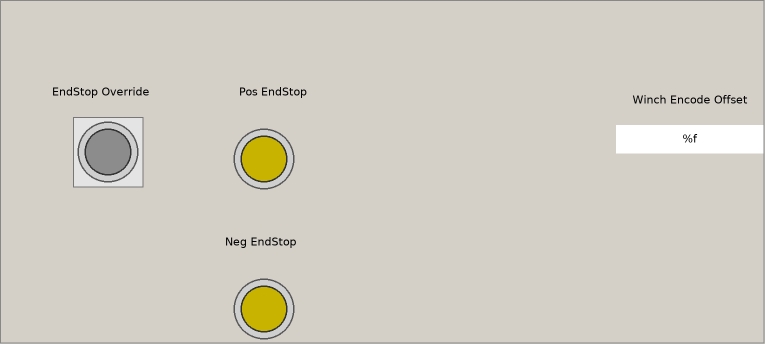
VISUALIZATION HMI  // 765x344
    PushSwitch (73,117 70x70), variable: HMI.bEndStopOverride, behaviour: TOGGLE, style: Switch-PushSwitch-Gray
    Lamp1 (229,124 70x70), variable: P_Outputs.bEndStopPosActive, style: Lamp-Lamp1-Yellow
    Label (26,77 150x30), "EndStop Override"
    Label (198,77 150x30), "Pos EndStop"
    Lamp1 (229,274 70x70), variable: P_Outputs.bEndStopNegActive, style: Lamp-Lamp1-Yellow
    Label (186,227 150x30), "Neg EndStop"
    Textfield (615,124 150x30), "%f", text variable: G_Parameters.stParam.fWinchEncoderOffset
        OnMouseClick: write the text variable via Default
    Label (615,85 150x30), "Winch Encode Offset"
END_VISUALIZATION

(* stored: Version 1.1.0.1, ProductVersion 3.1.4026.11
   Visu HMI: Id {7753864f-df6f-4a20-8851-17b344b9d768} *)
